ABB RobotStudio station: dispencing.rsstn

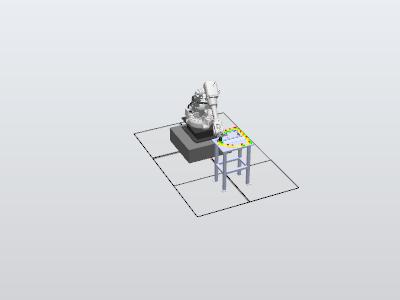
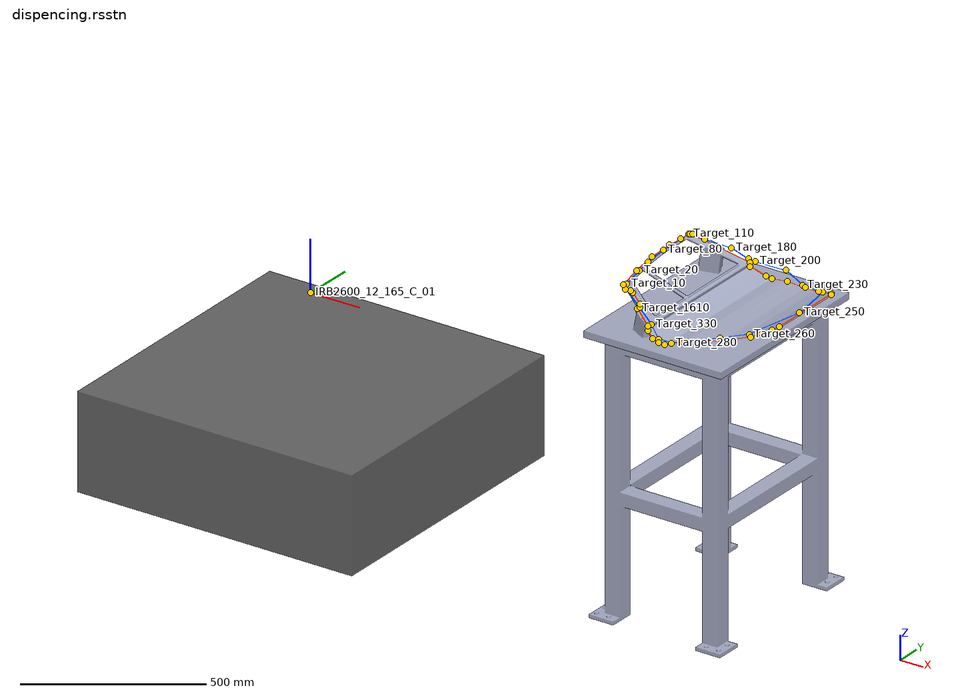
[picture v1: parts stored in the station drawn from their meshes, with robot base, taught points and paths (robot models come from the ABB library and are not in the file)]
Station Station (saved by RobotStudio 22.3.10141.1)
Controller dispencing, task T_ROB1: task frame (RAPID world) sits at (0, 0, 540) mm in the station
Controller dispencing
  mechanical unit ROB_1: IRB2600_12_165_C_01, 6 joints, base frame (0, 0, 0) mm
Layout (positions relative to the parent item):
  - IRB2600_12_165_C_01 [mechanism, from %ABB.RobotStudio.Models.IRB2600%\IRB2600_12_165_C_01.rslib] at (0, 0, 540) mm; joint values [-0.1944, 0.713, -0.0039, -0.0062, -0.2065, 0.0054] (rad or m)
  - Robotpedestal1400_H240_2 [part, from Equipment\Robot Pedestal 1400 H240.rslib] at (-30, 0, 300) mm
  - concrete [part] at (-450, -450, 0) mm, size 900 x 900 x 300 mm
  - Dispencer [mechanism, from Dispencing\Dispencer.rslib] at (1334.99, -262.8, 1043.19) mm, rotated rx 180 ry 61.2 rz 168.94 deg
  - table with door [part] at (1701.11, 257.98, 379.88) mm, rotated rx 90 ry 0 rz -90 deg, size 600 x 960.7 x 450 mm
Attachment: Dispencer is attached to IRB2600_12_165_C_01 / Link6
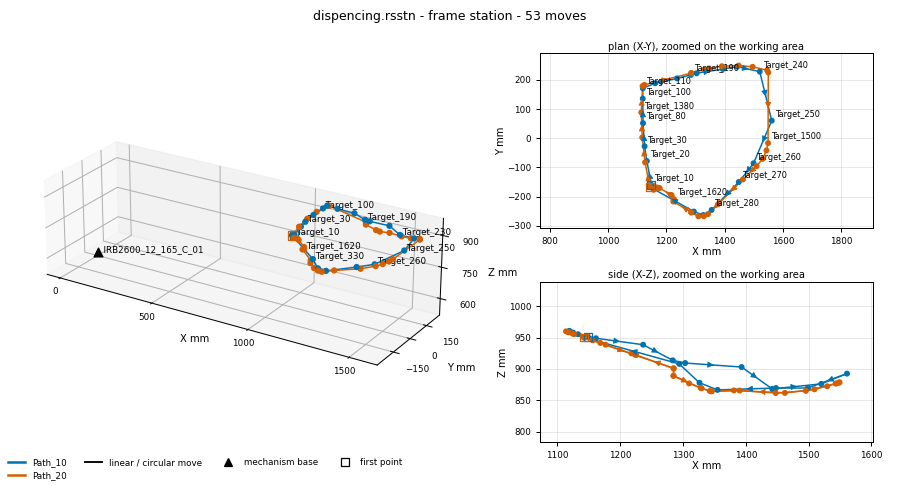
[picture p0: tool path of dispencing.rsstn in frame station, 53 of 53 moves have a stored position in this frame; points joined in program order, loops and branches not executed]
Targets, tools, work objects and paths stored in the station, written as RAPID:
! task T_ROB1
MODULE CalibData
  PERS tooldata Dispencer:=[TRUE,[[145,-0.097,55],[0.707106781,0,0.707106781,0]],[1,[0,0,1],[1,0,0,0],0,0,0]];
ENDMODULE

! task T_ROB1
MODULE Module1
  CONST robtarget Target_10:=[[1148.499962871,-159.971293351,411.314444863],[0.247506885,-0.093325063,-0.964083366,-0.0239591],[-1,0,-1,1],[9E+09,9E+09,9E+09,9E+09,9E+09,9E+09]];
  CONST robtarget Target_20:=[[1132.820949952,-78.089681396,415.265544379],[0.247506899,-0.093325059,-0.964083362,-0.023959132],[-1,0,-1,1],[9E+09,9E+09,9E+09,9E+09,9E+09,9E+09]];
  CONST robtarget Target_30:=[[1125.08998377,-27.474636398,417.837317978],[0.247506909,-0.093325075,-0.964083357,-0.023959153],[-1,0,-1,1],[9E+09,9E+09,9E+09,9E+09,9E+09,9E+09]];
  CONST robtarget Target_80:=[[1119.737967363,51.620353539,419.931160183],[0.247506891,-0.09332506,-0.964083365,-0.023959075],[0,0,-1,1],[9E+09,9E+09,9E+09,9E+09,9E+09,9E+09]];
  CONST robtarget Target_100:=[[1118.805032751,135.65229993,420.240228466],[0.247506904,-0.093325063,-0.964083362,-0.02395907],[0,0,-1,1],[9E+09,9E+09,9E+09,9E+09,9E+09,9E+09]];
  CONST robtarget Target_110:=[[1119.142039067,171.508992509,420.240231165],[0.247506902,-0.093325052,-0.964083363,-0.023959057],[0,0,-1,1],[9E+09,9E+09,9E+09,9E+09,9E+09,9E+09]];
  CONST robtarget Target_140:=[[1161.393030228,188.48850565,408.827210657],[0.247506909,-0.093324961,-0.964083369,-0.0239591],[0,0,-1,1],[9E+09,9E+09,9E+09,9E+09,9E+09,9E+09]];
  CONST robtarget Target_180:=[[1236.547614657,205.099344148,398.543162969],[0.247506911,-0.093324882,-0.964083374,-0.023959185],[0,0,-1,1],[9E+09,9E+09,9E+09,9E+09,9E+09,9E+09]];
  CONST robtarget Target_190:=[[1283.846009116,217.351587785,373.666905155],[0.2475069,-0.093324861,-0.96408338,-0.023959154],[0,0,-1,1],[9E+09,9E+09,9E+09,9E+09,9E+09,9E+09]];
  CONST robtarget Target_200:=[[1303.457010106,222.667097178,369.36726387],[0.247506912,-0.093324893,-0.964083372,-0.023959231],[0,0,-1,1],[9E+09,9E+09,9E+09,9E+09,9E+09,9E+09]];
  CONST robtarget Target_210:=[[1393.295031729,237.557131019,363.023179923],[0.247506898,-0.093324885,-0.964083376,-0.023959236],[0,0,-1,1],[9E+09,9E+09,9E+09,9E+09,9E+09,9E+09]];
  CONST robtarget Target_230:=[[1441.982641603,245.399770102,328.178619484],[0.247506907,-0.093324865,-0.964083375,-0.023959277],[0,0,-1,1],[9E+09,9E+09,9E+09,9E+09,9E+09,9E+09]];
  CONST robtarget Target_240:=[[1520.021774639,228.504869372,336.192420714],[0.247506909,-0.093324872,-0.964083373,-0.023959285],[0,1,-1,1],[9E+09,9E+09,9E+09,9E+09,9E+09,9E+09]];
  CONST robtarget Target_250:=[[1561.082216023,60.332298447,352.555111315],[0.24750691,-0.093324856,-0.964083375,-0.023959259],[0,1,-2,1],[9E+09,9E+09,9E+09,9E+09,9E+09,9E+09]];
  CONST robtarget Target_260:=[[1498.75698566,-85.86294228,329.602002811],[0.247506918,-0.093324844,-0.964083375,-0.023959255],[-1,0,-1,1],[9E+09,9E+09,9E+09,9E+09,9E+09,9E+09]];
  CONST robtarget Target_270:=[[1448.016984247,-150.190295263,329.602219559],[0.247506912,-0.09332485,-0.964083376,-0.023959246],[-1,0,-1,1],[9E+09,9E+09,9E+09,9E+09,9E+09,9E+09]];
  CONST robtarget Target_280:=[[1354.990949608,-245.835001369,326.64644037],[0.247506898,-0.093324847,-0.96408338,-0.02395924],[-1,0,-1,1],[9E+09,9E+09,9E+09,9E+09,9E+09,9E+09]];
  CONST robtarget Target_300:=[[1326.262943734,-263.475795665,337.942561218],[0.247506893,-0.093324845,-0.964083381,-0.023959238],[-1,-1,0,1],[9E+09,9E+09,9E+09,9E+09,9E+09,9E+09]];
  CONST robtarget Target_330:=[[1294.005979002,-251.292905757,368.011976552],[0.247506905,-0.093324846,-0.964083378,-0.02395924],[-1,0,-1,1],[9E+09,9E+09,9E+09,9E+09,9E+09,9E+09]];
  CONST robtarget Target_1050:=[[1142.798070581,-166.861822063,409.996200897],[0.12719091,-0.610260726,-0.775490891,0.100090946],[0,0,0,0],[9E+09,9E+09,9E+09,9E+09,9E+09,9E+09]];
  CONST robtarget Target_1350:=[[1142.798070581,-166.861822063,409.996200897],[0.12719091,-0.610260726,-0.775490891,0.100090946],[1,1,0,6],[9E+09,9E+09,9E+09,9E+09,9E+09,9E+09]];
  CONST robtarget Target_1360:=[[1126.770500444,-82.605001631,415.399011711],[0.123165212,-0.640222181,-0.75094596,0.105005027],[0,-2,1,0],[9E+09,9E+09,9E+09,9E+09,9E+09,9E+09]];
  CONST robtarget Target_1370:=[[1117.057563324,2.719130913,418.673192466],[0.118945019,-0.669228817,-0.725215185,0.109762504],[0,0,0,0],[9E+09,9E+09,9E+09,9E+09,9E+09,9E+09]];
  CONST robtarget Target_1380:=[[1113.724693123,88.456135157,419.796685735],[0.114545347,-0.69717683,-0.698390108,0.114346353],[0,0,0,0],[9E+09,9E+09,9E+09,9E+09,9E+09,9E+09]];
  CONST robtarget Target_1390:=[[1118.167114787,178.674994261,418.29916842],[0.078574022,-0.862725646,-0.4790707,0.14149858],[0,-2,0,2],[9E+09,9E+09,9E+09,9E+09,9E+09,9E+09]];
  CONST robtarget Target_1400:=[[1124.12409238,183.170931425,416.291102151],[0.018744458,-0.980174962,-0.114286126,0.160761843],[0,0,0,0],[9E+09,9E+09,9E+09,9E+09,9E+09,9E+09]];
  CONST robtarget Target_1410:=[[1285.124236156,223.23445932,360.853724302],[0.02118738,-0.863654725,-0.036428191,0.502319219],[0,0,0,0],[9E+09,9E+09,9E+09,9E+09,9E+09,9E+09]];
  CONST robtarget Target_1420:=[[1284.869348571,223.686738148,349.063750968],[0.027551853,-0.962782256,-0.10766825,0.246371204],[0,0,0,0],[9E+09,9E+09,9E+09,9E+09,9E+09,9E+09]];
  CONST robtarget Target_1430:=[[1329.598717961,235.070409919,329.16368642],[0.019417152,-0.979247572,-0.114460323,0.166120441],[0,0,0,0],[9E+09,9E+09,9E+09,9E+09,9E+09,9E+09]];
  CONST robtarget Target_1440:=[[1345.766627881,239.228445894,324.152655119],[0.005743891,0.992314812,0.112803089,0.050534976],[0,0,0,0],[9E+09,9E+09,9E+09,9E+09,9E+09,9E+09]];
  CONST robtarget Target_1450:=[[1390.149548943,246.959997305,325.580482045],[0.001089266,-0.998127208,-0.058244757,0.018666513],[0,0,0,0],[9E+09,9E+09,9E+09,9E+09,9E+09,9E+09]];
  CONST robtarget Target_1460:=[[1447.694229979,249.375878009,321.606149103],[0.000068104,0.999850014,-0.016840305,-0.00404349],[0,0,0,0],[9E+09,9E+09,9E+09,9E+09,9E+09,9E+09]];
  CONST robtarget Target_1470:=[[1495.645268603,244.831987746,325.111138427],[0.005840632,-0.994158865,0.075700484,-0.076703814],[0,0,0,0],[9E+09,9E+09,9E+09,9E+09,9E+09,9E+09]];
  CONST robtarget Target_1480:=[[1545.172613242,233.361979387,337.226164979],[0.048763152,-0.941094527,0.296721739,-0.154659161],[0,0,0,0],[9E+09,9E+09,9E+09,9E+09,9E+09,9E+09]];
  CONST robtarget Target_1490:=[[1549.240820427,225.492816496,338.633301557],[0.119715152,-0.696899187,0.696899048,-0.119714342],[0,0,0,0],[9E+09,9E+09,9E+09,9E+09,9E+09,9E+09]];
  CONST robtarget Target_1500:=[[1548.547017302,-16.624545395,338.388653922],[0.12536601,-0.656628541,0.735246257,-0.111960992],[0,0,0,0],[9E+09,9E+09,9E+09,9E+09,9E+09,9E+09]];
  CONST robtarget Target_1510:=[[1543.116843963,-41.911835799,336.540056928],[0.129075567,-0.573501553,0.803711592,-0.092103982],[0,0,0,0],[9E+09,9E+09,9E+09,9E+09,9E+09,9E+09]];
  CONST robtarget Target_1520:=[[1529.462923876,-70.804342011,332.398793715],[0.118692405,-0.470075403,0.872267008,-0.063964795],[0,0,0,0],[9E+09,9E+09,9E+09,9E+09,9E+09,9E+09]];
  CONST robtarget Target_1530:=[[1509.229214904,-95.541203694,327.544170819],[0.092994309,-0.367355064,0.924682397,-0.036942936],[0,0,0,0],[9E+09,9E+09,9E+09,9E+09,9E+09,9E+09]];
  CONST robtarget Target_1540:=[[1462.162010922,-141.434503019,321.841758711],[0.018805371,-0.379424029,0.924999601,-0.007713744],[0,0,0,0],[9E+09,9E+09,9E+09,9E+09,9E+09,9E+09]];
  CONST robtarget Target_1550:=[[1380.916137151,-222.423286842,325.792344478],[0.003924832,0.379376639,-0.925232604,-0.001609314],[0,0,0,0],[9E+09,9E+09,9E+09,9E+09,9E+09,9E+09]];
  CONST robtarget Target_1560:=[[1342.642729733,-260.035124085,324.942283009],[0.136758781,0.318415933,-0.936882036,-0.046479891],[0,0,0,0],[9E+09,9E+09,9E+09,9E+09,9E+09,9E+09]];
  CONST robtarget Target_1570:=[[1328.34588909,-267.39240962,329.604489914],[0.1680686,0.125859223,-0.977468202,-0.021640585],[0,0,0,0],[9E+09,9E+09,9E+09,9E+09,9E+09,9E+09]];
  CONST robtarget Target_1580:=[[1309.720555233,-267.861682155,336.919956861],[0.201496384,-0.100550541,-0.97409249,0.020799432],[0,0,0,0],[9E+09,9E+09,9E+09,9E+09,9E+09,9E+09]];
  CONST robtarget Target_1590:=[[1284.869254246,-254.898746298,349.063802561],[0.240271386,-0.239064943,-0.938815282,0.061183987],[0,0,0,0],[9E+09,9E+09,9E+09,9E+09,9E+09,9E+09]];
  CONST robtarget Target_1600:=[[1285.098404078,-253.68007029,360.898513338],[0.493798802,-0.107282557,-0.860735218,0.06154738],[0,0,0,0],[9E+09,9E+09,9E+09,9E+09,9E+09,9E+09]];
  CONST robtarget Target_1610:=[[1223.493918221,-217.082679742,382.794048949],[0.156474284,-0.25223889,-0.954033447,0.041370562],[0,0,0,0],[9E+09,9E+09,9E+09,9E+09,9E+09,9E+09]];
  CONST robtarget Target_1620:=[[1225.444463335,-208.698118808,382.136530301],[0.116459446,-0.685287076,-0.710060489,0.112396274],[0,0,0,0],[9E+09,9E+09,9E+09,9E+09,9E+09,9E+09]];
  CONST robtarget Target_1630:=[[1217.867847713,-195.499612709,384.690568154],[0.156474329,-0.252237858,-0.95403372,0.041370393],[0,0,0,0],[9E+09,9E+09,9E+09,9E+09,9E+09,9E+09]];
  CONST robtarget Target_1640:=[[1176.67871428,-170.787836484,398.575211528],[0.156474284,-0.252238889,-0.954033447,0.041370562],[0,0,0,0],[9E+09,9E+09,9E+09,9E+09,9E+09,9E+09]];
  CONST robtarget Target_1650:=[[1168.283328259,-168.753470862,401.405252638],[0.161764001,0.032339069,-0.986285182,-0.005304041],[0,0,0,0],[9E+09,9E+09,9E+09,9E+09,9E+09,9E+09]];
  CONST robtarget Target_1660:=[[1156.226416359,-176.724961561,405.469575233],[0.139897502,0.496243081,-0.852963702,-0.081390516],[0,0,0,0],[9E+09,9E+09,9E+09,9E+09,9E+09,9E+09]];
  CONST robtarget Target_1670:=[[1142.798070581,-166.861822063,409.996200897],[0.12719091,-0.610260727,-0.77549089,0.100090946],[0,0,0,0],[9E+09,9E+09,9E+09,9E+09,9E+09,9E+09]];
  PROC Path_10()
    MoveL Target_10,v1000,z100,Dispencer\WObj:=wobj0;
    MoveL Target_20,v1000,z100,Dispencer\WObj:=wobj0;
    MoveL Target_30,v1000,z100,Dispencer\WObj:=wobj0;
    MoveL Target_80,v1000,z100,Dispencer\WObj:=wobj0;
    MoveL Target_100,v1000,z100,Dispencer\WObj:=wobj0;
    MoveL Target_110,v1000,z100,Dispencer\WObj:=wobj0;
    MoveL Target_140,v1000,z100,Dispencer\WObj:=wobj0;
    MoveL Target_180,v1000,z100,Dispencer\WObj:=wobj0;
    MoveL Target_190,v1000,z100,Dispencer\WObj:=wobj0;
    MoveL Target_200,v1000,z100,Dispencer\WObj:=wobj0;
    MoveL Target_210,v1000,z100,Dispencer\WObj:=wobj0;
    MoveL Target_230,v1000,z100,Dispencer\WObj:=wobj0;
    MoveL Target_240,v1000,z100,Dispencer\WObj:=wobj0;
    MoveL Target_250,v1000,z100,Dispencer\WObj:=wobj0;
    MoveL Target_260,v1000,z100,Dispencer\WObj:=wobj0;
    MoveL Target_270,v1000,z100,Dispencer\WObj:=wobj0;
    MoveL Target_280,v1000,z100,Dispencer\WObj:=wobj0;
    MoveL Target_300,v1000,z100,Dispencer\WObj:=wobj0;
    MoveL Target_330,v1000,z100,Dispencer\WObj:=wobj0;
    MoveL Target_1050,v1000,z100,Dispencer\WObj:=wobj0;
  ENDPROC
  PROC Path_20()
    MoveL Target_1350,v1000,z100,Dispencer\WObj:=wobj0;
    MoveL Target_1360,v1000,z100,Dispencer\WObj:=wobj0;
    MoveL Target_1370,v1000,z100,Dispencer\WObj:=wobj0;
    MoveL Target_1380,v1000,z100,Dispencer\WObj:=wobj0;
    MoveL Target_1390,v1000,z100,Dispencer\WObj:=wobj0;
    MoveL Target_1400,v1000,z100,Dispencer\WObj:=wobj0;
    MoveL Target_1410,v1000,z100,Dispencer\WObj:=wobj0;
    MoveL Target_1420,v1000,z100,Dispencer\WObj:=wobj0;
    MoveL Target_1430,v1000,z100,Dispencer\WObj:=wobj0;
    MoveL Target_1440,v1000,z100,Dispencer\WObj:=wobj0;
    MoveL Target_1450,v1000,z100,Dispencer\WObj:=wobj0;
    MoveL Target_1460,v1000,z100,Dispencer\WObj:=wobj0;
    MoveL Target_1470,v1000,z100,Dispencer\WObj:=wobj0;
    MoveL Target_1480,v1000,z100,Dispencer\WObj:=wobj0;
    MoveL Target_1490,v1000,z100,Dispencer\WObj:=wobj0;
    MoveL Target_1500,v1000,z100,Dispencer\WObj:=wobj0;
    MoveL Target_1510,v1000,z100,Dispencer\WObj:=wobj0;
    MoveL Target_1520,v1000,z100,Dispencer\WObj:=wobj0;
    MoveL Target_1530,v1000,z100,Dispencer\WObj:=wobj0;
    MoveL Target_1540,v1000,z100,Dispencer\WObj:=wobj0;
    MoveL Target_1550,v1000,z100,Dispencer\WObj:=wobj0;
    MoveL Target_1560,v1000,z100,Dispencer\WObj:=wobj0;
    MoveL Target_1570,v1000,z100,Dispencer\WObj:=wobj0;
    MoveL Target_1580,v1000,z100,Dispencer\WObj:=wobj0;
    MoveL Target_1590,v1000,z100,Dispencer\WObj:=wobj0;
    MoveL Target_1600,v1000,z100,Dispencer\WObj:=wobj0;
    MoveL Target_1610,v1000,z100,Dispencer\WObj:=wobj0;
    MoveL Target_1620,v1000,z100,Dispencer\WObj:=wobj0;
    MoveL Target_1630,v1000,z100,Dispencer\WObj:=wobj0;
    MoveL Target_1640,v1000,z100,Dispencer\WObj:=wobj0;
    MoveL Target_1650,v1000,z100,Dispencer\WObj:=wobj0;
    MoveL Target_1660,v1000,z100,Dispencer\WObj:=wobj0;
    MoveL Target_1670,v1000,z100,Dispencer\WObj:=wobj0;
  ENDPROC
ENDMODULE

